PROGRAM MAIN
VAR

	
	
END_VAR



AXES_CYCLE();
PIST_CYCLE();
STATION_CYCLE();

END_PROGRAM

(* stored: Version 1.1.0.1, ProductVersion 3.1.4024.12
   POU MAIN: Id {6c7239d6-f7f9-4e71-8a46-bf89f21a2b56}, SpecialFunc None *)
